FUNCTION_BLOCK FB_FanControl
VAR_INPUT
	fSpeed	:	REAL;		//Fan speed setpoint 0..100%
END_VAR
VAR
	fSpeedSetRaw  AT%Q*	: INT 	:=0; 	//Raw value for terminal => send to valve
END_VAR
VAR CONSTANT
		fFactor : REAL :=327.67;	// factor for calculating the terminal integer values (from percentage to int)
END_VAR

fSpeedSetRaw := REAL_TO_INT(fSpeed*fFactor);

END_FUNCTION_BLOCK

(* stored: Version 1.1.0.1, ProductVersion 3.1.4024.9
   POU FB_FanControl: Id {2862505f-0eab-4e09-abf3-83a637c0182e}, SpecialFunc None *)
